INTERFACE I_HaveErrors EXTENDS __SYSTEM.IQueryInterface

METHOD AddError
VAR_INPUT
	ErrorToAdd : I_Error;
END_VAR
END_METHOD

METHOD PUBLIC GetErrors : I_ErrorCollection
VAR_INPUT
END_VAR
END_METHOD

END_INTERFACE

(* stored: Version 1.1.0.1, ProductVersion 3.1.4024.12
   Itf I_HaveErrors: Id {6c14ee43-6ab7-0c30-3bf7-4a331785d2fc}
   Method AddError: Id {23aee699-1229-0461-1c27-f5ff339c8835}
   Method GetErrors: Id {08c9815a-9cf4-0ac6-3683-4e6b7fc0ea52} *)
